Universal Robots PolyScope program: mm_start.urp

Program mm_start (installation=default directory=/programs createdIn=5.19.0 lastSavedIn=5.19.0 robotSerialNumber=20245203260)
Calibrated DH parameters: a=[0.00002, -0.297909, -0.550376, -0.000026, 0.000029, 0]; d=[0.180392, 372.242289, -404.966968, 32.898661, 0.119952, 0.115576]; alpha=[1.570137, -0.001437, 0.004676, 1.569919, -1.569683, 0]; deltaTheta=[0, -1.062765, 0.791609, 0.271161, 0, 0]
InitVariablesNode
Robot Program (runOnlyOnce=false)
  MoveJ speed 60 deg/s, acceleration 80 deg/s^2 (useActiveTCP=true) feature=Base
    Waypoint MM_Home: TCP in base x=118.127 y=-551.155 z=1157.021 mm, rx=0.0072 ry=-0.0069 rz=-0.0037 rad; joints [84.243, -100.906, 79.201, -67.911, 90.606, 5.632] deg; TCP offset x=0 y=0 z=50 mm, rx=0 ry=0 rz=0 rad
